FUNCTION_BLOCK ConveyorEntry
VAR_INPUT
END_VAR
VAR_OUTPUT
END_VAR
VAR
	ConveyorEntryToken : INT;
END_VAR

//If emergency button is activated or system isn't started or stopped, reset system token to 10.
IF NOT SystemStarted OR EmergencyActivated THEN
	ConveyorEntryToken := 10;
END_IF
//Conveyor entry system conditions.
CASE ConveyorEntryToken OF
	//
	10:
		//Waiting for system start
		IF SystemStarted THEN
			ConveyorEntryToken := 20;
		END_IF
	20:
		//Start conveyor entry motor when system is started. Continue to work until pallet is loaded or if loaded already , work until pallet sensor activates.
		Conveyor_Entry := TRUE;
		IF TransferBusy AND Pallet_Sensor THEN
			ConveyorEntryToken := 30;
		ELSIF NOT TransferBusy AND Loaded THEN
			ConveyorEntryToken := 30;
		END_IF
	30:
		//Stop until pallet is pushed one side completely. 
		Conveyor_Entry := FALSE;
		IF NOT TransferBusy AND NOT Loaded THEN
			ConveyorEntryToken := 20;
		END_IF
ELSE
	ConveyorEntryToken := 10;
END_CASE

END_FUNCTION_BLOCK

(* stored: Version 1.1.0.1, ProductVersion 3.1.4024.6
   POU ConveyorEntry: Id {5d697ee2-3acb-4ff2-bd79-036fcf3678d1}, SpecialFunc None *)
